FUNCTION_BLOCK fb_Blink
VAR_INPUT
	tLowTime		: TIME;
	tCycleTime	: TIME;
END_VAR
VAR_OUTPUT
	bCycle			: BOOL;
END_VAR
VAR
	tonLowTime		: TON;
	tofCycleTime	: TOF;
END_VAR

tonLowTime(IN:=(NOT tofCycleTime.Q), PT:= tLowTime);
tofCycleTime(IN:=(tonLowTime.Q), PT:= tCycleTime);

bCycle := tofCycleTime.Q;

END_FUNCTION_BLOCK

(* stored: Version 1.1.0.1, ProductVersion 3.1.4022.16
   POU fb_Blink: Id {87a5ec5a-f5e6-4edf-8c00-afb3fd9280e0}, SpecialFunc None *)
